// Mitsubishi GX Developer project: Ножницы(гильотина) №5   PLC: FX3G

PROGRAM MAIN
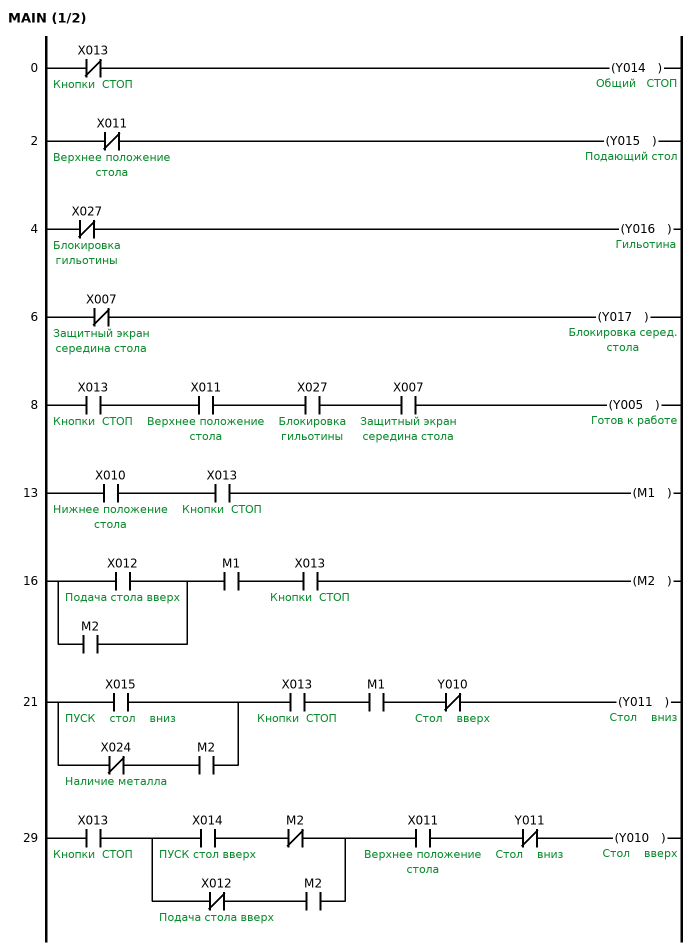
0     LDI     X013  ; Кнопки  СТОП
      OUT     Y014  ; Общий   СТОП
2     LDI     X011  ; Верхнее положение стола
      OUT     Y015  ; Подающий стол
4     LDI     X027  ; Блокировка гильотины
      OUT     Y016  ; Гильотина
6     LDI     X007  ; Защитный экран середина стола
      OUT     Y017  ; Блокировка серед. стола
8     LD      X013  ; Кнопки  СТОП
      AND     X011  ; Верхнее положение стола
      AND     X027  ; Блокировка гильотины
      AND     X007  ; Защитный экран середина стола
      OUT     Y005  ; Готов к работе
13    LD      X010  ; Нижнее положение стола
      AND     X013  ; Кнопки  СТОП
      OUT     M1
16    LD      X012  ; Подача стола вверх
      OR      M2
      AND     M1
      AND     X013  ; Кнопки  СТОП
      OUT     M2
21    LD      X015  ; ПУСК    стол    вниз
      LDI     X024  ; Наличие металла
      AND     M2
      ORB
      AND     X013  ; Кнопки  СТОП
      AND     M1
      ANI     Y010  ; Стол    вверх
      OUT     Y011  ; Стол    вниз
29    LD      X013  ; Кнопки  СТОП
      LD      X014  ; ПУСК стол вверх
      ANI     M2
      LDI     X012  ; Подача стола вверх
      AND     M2
      ORB
      ANB
      AND     X011  ; Верхнее положение стола
      ANI     Y011  ; Стол    вниз
      OUT     Y010  ; Стол    вверх
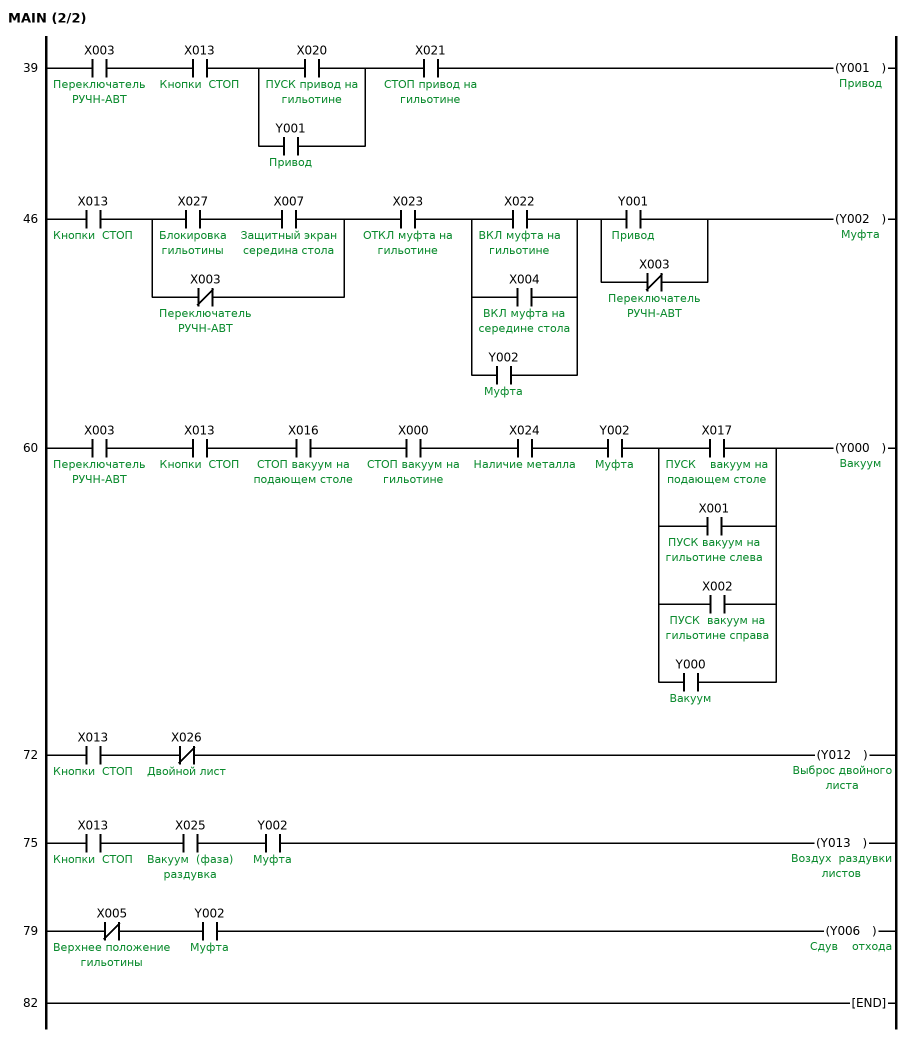
39    LD      X003  ; Переключатель   РУЧН-АВТ
      AND     X013  ; Кнопки  СТОП
      LD      X020  ; ПУСК привод на гильотине
      OR      Y001  ; Привод
      ANB
      AND     X021  ; СТОП привод на гильотине
      OUT     Y001  ; Привод
46    LD      X013  ; Кнопки  СТОП
      LD      X027  ; Блокировка гильотины
      AND     X007  ; Защитный экран середина стола
      ORI     X003  ; Переключатель   РУЧН-АВТ
      ANB
      AND     X023  ; ОТКЛ муфта на гильотине
      LD      X022  ; ВКЛ муфта на гильотине
      OR      X004  ; ВКЛ муфта на середине стола
      OR      Y002  ; Муфта
      ANB
      LD      Y001  ; Привод
      ORI     X003  ; Переключатель   РУЧН-АВТ
      ANB
      OUT     Y002  ; Муфта
60    LD      X003  ; Переключатель   РУЧН-АВТ
      AND     X013  ; Кнопки  СТОП
      AND     X016  ; СТОП вакуум на подающем столе
      AND     X000  ; СТОП вакуум на гильотине
      AND     X024  ; Наличие металла
      AND     Y002  ; Муфта
      LD      X017  ; ПУСК    вакуум на подающем столе
      OR      X001  ; ПУСК вакуум на  гильотине слева
      OR      X002  ; ПУСК  вакуум на гильотине справа
      OR      Y000  ; Вакуум
      ANB
      OUT     Y000  ; Вакуум
72    LD      X013  ; Кнопки  СТОП
      ANI     X026  ; Двойной лист
      OUT     Y012  ; Выброс двойного листа
75    LD      X013  ; Кнопки  СТОП
      AND     X025  ; Вакуум  (фаза) раздувка
      AND     Y002  ; Муфта
      OUT     Y013  ; Воздух  раздувки листов
79    LDI     X005  ; Верхнее положение гильотины
      AND     Y002  ; Муфта
      OUT     Y006  ; Сдув    отхода
82    END
END_PROGRAM
